TYPE CAN_MsgSlot :
STRUCT
	cobId : UINT; // Unsigned 16-bit
    data  : ARRAY[0..7] OF BYTE;
END_STRUCT
END_TYPE

(* stored: Version 1.1.0.1
   DUT CAN_MsgSlot: Id {e2d4410a-4abe-4a2a-8e75-cbf1e294c437} *)
